RoboDK station: RDK_program.rdk

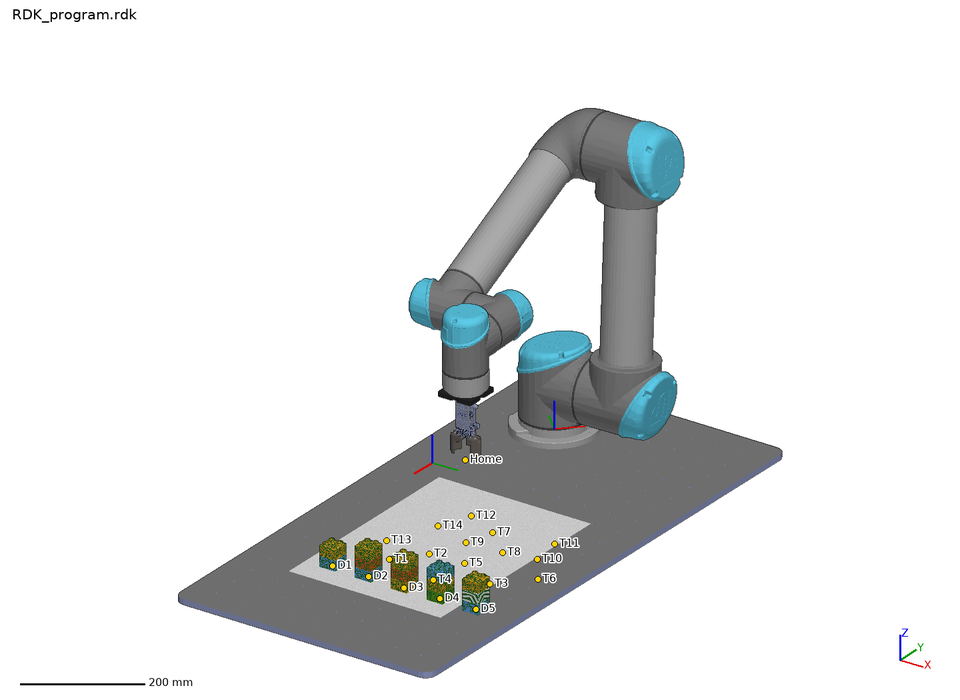
[picture v0: the station drawn from its stored meshes, robots at their saved joint values, targets as dots, program paths as lines]
Station RDK_program (saved by RoboDK 5.4.1). Poses are relative to the parent item; angles as X-Y-Z fixed-axis rotations.
  - frame UR5 Base at (0, 0, 0) mm, rotated rx 0 ry 0 rz 45 deg
    - robot UR5: 6 axes, payload 5 kg, reach 850 mm, repeatability 0.1 mm, weight 18.4 kg
        modified DH rows (alpha deg, a mm, theta deg, d mm): 0, 0, 0, 89.2; 90, 0, 180, 0; 0, 425, 0, 0; 0, 392.43, 0, 109; -90, 0, 0, 93.65; 90, 0, 180, 82
        joint limits [-360, -360, -360, -360, -360, -360] to [360, 360, 360, 360, 360, 360]; home [0, -90, -90, 0, 90, 0]; saved at [47.127, -93.093, 116.518, -113.505, -89.821, -177.881]
      - tool gripper_full_2, TCP at (0, 0, 116) mm, rotated rx 180 ry 0 rz 0 deg, size 65 x 113.3 x 65 mm, geometry from gripper_full_2.STEP
    - object Tabletop3 at (0, 0, -10) mm, rotated rx 0 ry 0 rz -135 deg, size 1000 x 500 x 10.1 mm, geometry from Tabletop3.STEP
    - target Home (joint target) at (-212.95, -390.53, 150.71) mm, rotated rx -0.07 ry -0.18 rz -44.99 deg; joints [47.127, -93.093, 116.518, -113.505, -89.821, -177.881] of UR5
  - Python program Prog1 (listed below)
  - frame Reference at (-89, -213, 0) mm, rotated rx 0 ry 0 rz -90 deg
    - target D1 (Cartesian target) at (400, 85, 0) mm, rotated rx 0 ry 0 rz 45 deg; joints [-39.774, -124.478, -93.696, -51.826, 90, -129.774] of UR5
    - target D2 (Cartesian target) at (400, 155, 0) mm, rotated rx 0 ry 0 rz 45 deg; joints [-33.151, -124.323, -93.972, -51.705, 90, -123.151] of UR5
    - target D3 (Cartesian target) at (400, 225, 0) mm, rotated rx 0 ry 0 rz 45 deg; joints [-26.713, -125.097, -92.593, -52.31, 90, -116.713] of UR5
    - target D4 (Cartesian target) at (400, 295, 0) mm, rotated rx 0 ry 0 rz 45 deg; joints [-20.613, -126.788, -89.555, -53.657, 90, -110.613] of UR5
    - target D5 (Cartesian target) at (400, 365, 0) mm, rotated rx 0 ry 0 rz 45 deg; joints [-14.958, -129.386, -84.831, -55.783, 90, -104.958] of UR5
    - target T1 (Cartesian target) at (329.2, 146.4, 0) mm, rotated rx 0 ry 0 rz 45 deg; joints [49.602, -72.102, -157.001, -40.897, 90, 3.602] of UR5
    - target T2 (Cartesian target) at (276.1, 187.4, 0) mm, rotated rx 0 ry 0 rz -45 deg; joints [188.195, -85.112, -221.34, 36.452, 90, 82.195] of UR5
    - target T3 (Cartesian target) at (309.7, 329.1, 0) mm, rotated rx 0 ry 0 rz 34 deg; joints [137.212, -81.175, -226.125, 37.3, 90, 26.212] of UR5
    - target T4 (Cartesian target) at (349.6, 247.2, 0) mm, rotated rx 0 ry 0 rz -3 deg; joints [117.872, -76.15, -232.881, 39.031, 90, 56.872] of UR5
    - target T5 (Cartesian target) at (270.7, 252.4, 0) mm, rotated rx 0 ry 0 rz -43 deg; joints [141.49, -81.14, -226.169, 37.309, 90, 31.49] of UR5
    - target T6 (Cartesian target) at (252.4, 383.1, 0) mm, rotated rx 0 ry 0 rz -42 deg; joints [51.9, -28.881, -165.501, -75.618, 90, -59.1] of UR5
    - target T7 (Cartesian target) at (154.7, 225.8, 0) mm, rotated rx 0 ry 0 rz 26 deg; joints [2.495, -82.844, -150.273, -36.883, 90, -86.505] of UR5
    - target T8 (Cartesian target) at (205.4, 281.4, 0) mm, rotated rx 0 ry 0 rz 37 deg; joints [116.931, -93.16, -213.07, 36.23, 90, 48.931] of UR5
    - target T9 (Cartesian target) at (208.6, 212.3, 0) mm, rotated rx 0 ry 0 rz -35 deg; joints [42.375, -60.732, -161.339, -47.93, 90, -17.625] of UR5
    - target T10 (Cartesian target) at (193.9, 340.5, 0) mm, rotated rx 0 ry 0 rz 20 deg; joints [102.889, -90.694, -215.384, 36.078, 90, -24.111] of UR5
    - target T11 (Cartesian target) at (131.5, 330.6, 0) mm, rotated rx 0 ry 0 rz -42 deg; joints [51.692, -75.106, -155.42, -39.474, 90, -60.308] of UR5
    - target T12 (Cartesian target) at (123.7, 162.9, 0) mm, rotated rx 0 ry 0 rz 6 deg; joints [63.3, -60.586, -161.38, -48.034, 90, 11.3] of UR5
    - target T13 (Cartesian target) at (274.7, 102.3, 0) mm, rotated rx 0 ry 0 rz -28 deg; joints [15.588, -74.336, -155.845, -39.818, 90, -98.412] of UR5
    - target T14 (Cartesian target) at (183.4, 139.4, 0) mm, rotated rx 0 ry 0 rz 27 deg; joints [15.174, -65.624, -159.754, -44.622, 90, -68.826] of UR5
  - object Duplo1 at (-4, -613, 0) mm, rotated rx 90 ry 0 rz -45 deg, size 44.4 x 23.7 x 44.4 mm, geometry from Duplo.STEP
  - object Duplo5 at (-4, -613, 19.2) mm, rotated rx 90 ry 0 rz -45 deg, size 44.4 x 23.7 x 44.4 mm, geometry from Duplo.STEP
  - object Duplo2 at (66, -613, 0) mm, rotated rx 90 ry 0 rz -45 deg, size 44.4 x 23.7 x 44.4 mm, geometry from Duplo.STEP
  - object Duplo11 at (66, -613, 19.2) mm, rotated rx 90 ry 0 rz -45 deg, size 44.4 x 23.7 x 44.4 mm, geometry from Duplo.STEP
  - object Duplo6 at (66, -613, 38.4) mm, rotated rx 90 ry 0 rz -45 deg, size 44.4 x 23.7 x 44.4 mm, geometry from Duplo.STEP
  - object Duplo7 at (136, -613, 0) mm, rotated rx 90 ry 0 rz -45 deg, size 44.4 x 23.7 x 44.4 mm, geometry from Duplo.STEP
  - object Duplo12 at (136, -613, 19.2) mm, rotated rx 90 ry 0 rz -45 deg, size 44.4 x 23.7 x 44.4 mm, geometry from Duplo.STEP
  - object Duplo8 at (136, -613, 38.4) mm, rotated rx 90 ry 0 rz -45 deg, size 44.4 x 23.7 x 44.4 mm, geometry from Duplo.STEP
  - object Duplo13 at (206, -613, 0) mm, rotated rx 90 ry 0 rz -45 deg, size 44.4 x 23.7 x 44.4 mm, geometry from Duplo.STEP
  - object Duplo9 at (206, -613, 19.2) mm, rotated rx 90 ry 0 rz -45 deg, size 44.4 x 23.7 x 44.4 mm, geometry from Duplo.STEP
  - object Duplo3 at (206, -613, 38.4) mm, rotated rx 90 ry 0 rz -45 deg, size 44.4 x 23.7 x 44.4 mm, geometry from Duplo.STEP
  - object Duplo4 at (276, -613, 0) mm, rotated rx 90 ry 0 rz -45 deg, size 44.4 x 23.7 x 44.4 mm, geometry from Duplo.STEP
  - object Duplo14 at (276, -613, 19.2) mm, rotated rx 90 ry 0 rz -45 deg, size 44.4 x 23.7 x 44.4 mm, geometry from Duplo.STEP
  - object Duplo10 at (276, -613, 38.4) mm, rotated rx 90 ry 0 rz -45 deg, size 44.4 x 23.7 x 44.4 mm, geometry from Duplo.STEP

--- Python program Prog1 ---
from robodk.robolink import *       # Import the robolink library (bridge with RoboDK)
from robodk.robomath import *       # Import the robomath library
from robodk.robofileio import *     # Import the robofile io file operation toolbox

RDK = Robolink()                    # establish a link with the simulator
robot = RDK.Item('UR5')             # retrieve the robot by name
tool = RDK.Item('gripper_full_2')   # Retrieve tool item
home = RDK.Item('home')             # Retrieve home item

h = 19.2                        # Height of LEGO brick w/o studs
ApDist = 5*h                    # Desired approach distance on pickup
buildCounter = 5                # Number of builds

RefPose = transl(-89,-213,0)*rotz(3/2*pi)   # Position of reference coordinate system

DelPose1 = transl(400,85,0)*rotz(pi/4)      # Build positions for Simpsons family
DelPose2 = transl(400,155,0)*rotz(pi/4)
DelPose3 = transl(400,225,0)*rotz(pi/4)
DelPose4 = transl(400,295,0)*rotz(pi/4)
DelPose5 = transl(400,365,0)*rotz(pi/4)

# Color sequence of each build
fig1 = ['blue', 'yellow']
fig2 = ['blue','orange','yellow']
fig3 = ['yellow','orange','yellow']
fig4 = ['green','yellow','blue']
fig5 = ['blue','white','yellow']


targets = []                # Empty target array
targetPoses = []            # Empty target poses array
bricks = []                 # Empty brick array
deliv = []                  # Empty delivery array

colors = fig1 + fig2 + fig3 + fig4 + fig5           # Array of color sequence for the builds

heights = [len(fig1), len(fig2), len(fig3),
           len(fig4), len(fig5)]                    # Array of heights for the builds

DelPose = [DelPose1, DelPose2, DelPose3, DelPose4, DelPose5] # Array of build positions

Reference = RDK.Item('Reference')       # Retrieve reference item
Reference.setPose(RefPose)              # Set pose of reference item real-life position

robot.setPoseFrame(Reference)       # Set frame of robot to reference frame

# Import csv file with real-life brick information from vision
path = 'C:\\Users\\esben\\OneDrive - Aalborg Universitet\\VT2 Welltec\\Robot Vision Miniprojekt TOP SECRET\\Python code\\'
import csv
with open(path+'bricks_data.csv', newline= '\n') as csvfile:
    Pos = list(csv.reader(csvfile))     # Save vision data in array
for i in range(len(Pos)):
    for j in range(5):
        try:
            Pos[i][j] = float(Pos[i][j])
        except Exception:
            pass

itemCounter = len(Pos)      # Number of LEGO bricks

# Define search function with input desired color and array of positions
def search(color, data_array):
    for j, brick in enumerate(data_array):
        if brick[3] == color and brick[4] == 0:             # If color = desired and it has not been used
            data_array[j][4] = 1                            # Set as used
            return brick[0],brick[1],brick[2],brick[3]      # Return X, Y, orientation, color

    return -1

for i in range(buildCounter):
    deliv.append(RDK.Item('D' + str(i + 1)))    # Retrieve build items in 'deliv' array
    deliv[i].setParent(Reference)               # Set reference coordinate system as parent of build items
    deliv[i].setPose(DelPose[i])                # Set desired position of build item

for i in range(itemCounter):
    targets.append(RDK.Item('T'+str(i+1)))      # Retrieve target items in 'targets' array
    Y,X,rot,col = search(colors[i],Pos)         # Search for i'th desired color and retrieve coordinates and orientation
    targets[i].setParent(Reference)             # Set reference coordinate system as parent of target item

    targets[i].setPose(transl(X,Y,0)*rotz(-rot+(pi/4)))     # Set pose of targets to coordinates/orientation of brick
    targetPoses.append(targets[i].Pose())                   # Retrieve target positions in 'targetPoses' array

# Define additional search function for placing virtual bricks in RoboDK (identical to previous)
def search1(color, data_array):
    for j, brick in enumerate(data_array):
        if brick[3] == color and brick[4] == 1:             # If color = desired and it has not been used
            data_array[j][4] = 2                            # Set as used
            return brick[0],brick[1],brick[2],brick[3]      # Return X, Y, orientation, color

    return -1

# Colors of virtual bricks for simulation representation
colorRef = ['blue','blue','blue','blue',
            'yellow','yellow','yellow','yellow','yellow','yellow',
            'orange','orange','green','white']

for i in range(itemCounter):
    bricks.append(RDK.Item('Duplo'+str(i+1)))   # Retrieve brick items in 'bricks' array
    Y, X, rot, col = search1(colorRef[i], Pos)  # Search for first desired brick item and retrieve corresponding coordinates/orientation
    bricks[i].setParent(Reference)              # Set reference coordinate system as parent of brick item
    bricks[i].setPose(transl(X, Y, 0) * rotz(-rot+(pi/4))*rotx(pi/2))  # Set pose of brick items to coordinates of real-life brick

for i in range(itemCounter):
    approach = targetPoses[i]*transl(0,0,ApDist)         # Set approach distance
    depart = targetPoses[i]*transl(0,0,ApDist)           # Set departure distance

    robot.setDO(0, 1)
    robot.setDO(1, 0)           # Open gripper

    robot.MoveL(approach)       # Move to brick approach position
    robot.MoveL(targets[i])     # Move to target

    tool.AttachClosest()        # Attach brick (in simulation)
    robot.setDO(0, 0)
    robot.setDO(1, 1)           # Close gripper

    robot.Pause(250)            # Wait 250 ms

    robot.MoveL(depart)         # Move to brick departure position

    if i <= heights[0]-1:           # If first build

        approachDeliv = deliv[0].Pose()*transl(0,0,ApDist)                  # set build approach
        deliver = deliv[0].Pose()*transl(0,0,(i*h))                         # set build position

    elif i <= sum(heights[0:2])-1:  # If second build

        approachDeliv = deliv[1].Pose()*transl(0,0,ApDist)                  # set build approach
        deliver = deliv[1].Pose()*transl(0,0,((i-sum(heights[0:1]))*h))     # set build position

    elif i <= sum(heights[0:3])-1:  # If third build

        approachDeliv = deliv[2].Pose()*transl(0,0,ApDist)                  # set build approach
        deliver = deliv[2].Pose()*transl(0,0,((i-sum(heights[0:2]))*h))     # set build position

    elif i <= sum(heights[0:4])-1:  # If fourth build

        approachDeliv = deliv[3].Pose()*transl(0,0,ApDist)                  # set build approach
        deliver = deliv[3].Pose()*transl(0,0,((i-sum(heights[0:3]))*h))     # set build position

    else:                           # If last build

        approachDeliv = deliv[4].Pose()*transl(0,0,ApDist)                  # set build approach
        deliver = deliv[4].Pose()*transl(0,0,((i-sum(heights[0:4]))*h))     # set build position

    robot.MoveL(approachDeliv)          # Move to build approach
    robot.MoveL(deliver)                # Move to build point

    tool.DetachAll()                    # Detach brick
    robot.setDO(0, 1)
    robot.setDO(1, 0)                   # Open gripper

    robot.Pause(250)                    # Wait 250 ms

    robot.MoveL(approachDeliv)          # Move to build departure

    if i == itemCounter-1:      # If last build is complete
        robot.MoveJ(home)       # Move home
    else:
        continue
